FUNCTION_BLOCK CfbOneLink
  (* Standard: 61499-2 *)
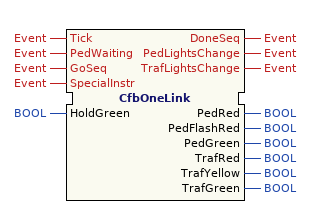
  EVENT_INPUT
    Tick;
    PedWaiting;
    GoSeq;
    SpecialInstr;
  END_EVENT
  EVENT_OUTPUT
    DoneSeq;
    PedLightsChange;
    TrafLightsChange;
  END_EVENT
  VAR_INPUT
    HoldGreen : BOOL;
  END_VAR
  VAR_OUTPUT
    PedRed : BOOL;
    PedFlashRed : BOOL;
    PedGreen : BOOL;
    TrafRed : BOOL;
    TrafYellow : BOOL;
    TrafGreen : BOOL;
  END_VAR
  FBS
    ped : BfbOnePedCtrl;
    traf : BfbOneWayCtrl;
  END_FBS
  EVENT_CONNECTIONS
    Tick TO ped.Tick;
    Tick TO traf.Tick;
    GoSeq TO traf.BeginSeq;
    traf.DoneSeq TO DoneSeq;
    PedWaiting TO ped.PedWaiting;
    traf.PedGrant TO ped.SeqGrant;
    ped.SeqStatusChange TO traf.PedStatusChange;
    SpecialInstr TO traf.SpecialInstr;
    ped.LightCtrlChange TO PedLightsChange;
    traf.LightCtrlChange TO TrafLightsChange;
  END_CONNECTIONS
  DATA_CONNECTIONS
    ped.Running TO traf.PedRunning;
    ped.Request TO traf.PedRequest;
    HoldGreen TO traf.HoldGreen;
    ped.LightRed TO PedRed;
    ped.LightFlashRed TO PedFlashRed;
    ped.LightGreen TO PedGreen;
    traf.LightRed TO TrafRed;
    traf.LightYellow TO TrafYellow;
    traf.LightGreen TO TrafGreen;
  END_CONNECTIONS
END_FUNCTION_BLOCK
